// TIA Portal V20 export
DATA_BLOCK "CallEquipment_DB"   // DB76
{ DB_Accessible_From_OPC_UA := 'FALSE' }
// stored: AssignedProDiagFB Unit1.Em1.ProDiag, DBAccessibleFromOPCUA false, DBAccessibleFromWebserver false, InstanceOfName Unit1.Em1.CallEquipment, InstanceOfType FB, Namespace Unit1.Em1
"Unit1.Em1.CallEquipment"
   // VAR_INPUT
   //    ZoneOperationEnable { ExternalWritable := 'False'} : "LWONIK_typeSafetyZoneManualOperation";
   //    unitEnableControlInterfaces { ExternalWritable := 'False'} : "LAF_typeEnableControlInterfaces";
   //    commandExcute { ExternalWritable := 'False'} : Bool;
   // END_VAR
   // VAR_IN_OUT
   //    unitStatus : "LAF_typeUnitStatus";
   //    emFeedback : "LUC_typeEmFeedback";
   //    unitAlarmDB : "LAF_typeAlarms";
   // END_VAR
   // VAR
   //    instSequenceUnWinder { ExternalWritable := 'False'} : "Unit1.Em1.Sequence_1_UnWinder";
   //    instUnWinderInitializedJob1 { ExternalWritable := 'False'} : "LAF_SelectJob";
   //    instUnWinderRunJob2 { ExternalWritable := 'False'} : "LAF_SelectJob";
   //    instUnWinderStopJob3 { ExternalWritable := 'False'} : "LAF_SelectJob";
   //    instUnWinderRewindJob4 { ExternalWritable := 'False'} : "LAF_SelectJob";
   //    instCmUnWinderAxisB { ExternalWritable := 'False'} : "LBC_AxisControl_TecPlcCn";
   //    instCmAirShaftOnOff { ExternalWritable := 'False'} : "LBC_TwoWayActuatorCn";
   //    instcmExpelFwdBwd { ExternalWritable := 'False'} : "LBC_TwoWayActuatorCn";
   //    instCmTensionCheckSensor { ExternalWritable := 'False'} : "LBC_DigitalSignalCn";
   //    instCmRadiusMeasureAnalogInput { ExternalWritable := 'False'} : "LBC_AnalogInputCn";
   //    instCmEpc { ExternalWritable := 'False'} : "LER_EPC_CON600";
   //    instCmRadiusMeasure { ExternalWritable := 'False'} : "LER_RadiusMeasure";
   //    instUnWinderAxisControlInterlockSummary { ExternalWritable := 'False'} : "LER_AxisControl_InterlockSummary";
   //    instServoTorqueCal_DR2 { ExternalWritable := 'False'} : "LER_ServoTorqueCal";
   //    instLDrv701ControlUnWinderAxisB { ExternalWritable := 'False'} : "LDrvSafe_SinaTlg701Control";
   //    instLDrv701StatusUnWinderAxisB { ExternalWritable := 'False'} : "LDrvSafe_SinaTlg701Status";
   //    statUnitStatus { ExternalWritable := 'False'} : "LAF_typeUnitStatus";
   //    statAllBrakeTest { ExternalWritable := 'False'} : "LER_typeBrakeTestUnitCommands";
   //    instManageAlarms { ExternalWritable := 'False'} : "LAF_ManageAlarms";
   //    instEventsPFE { S7_SetPoint := 'True'} : "Unit1.Em1.EventsPFE";
   //    statEnableManualCmds { ExternalWritable := 'False'} : Bool;
   //    statRcEnableCmds { ExternalWritable := 'False'} : Bool;
   //    statPulse { ExternalWritable := 'False'} : Array[0..99] of Bool;
   //    statTonTimer { ExternalWritable := 'False'} : Array[0..99] of TON_TIME;
   //    statTofTimer { ExternalWritable := 'False'} : Array[0..99] of TOF_TIME;
   //    statRadius { ExternalWritable := 'False'} : LReal;
   //    statDiameter { ExternalWritable := 'False'} : LReal;
   //    citi_Ptrig : Array[0..20] of Bool;
   //    citiTon : Array[0..20] of TON_TIME;
   //    citi : Time;
   //    citiTest : Array[0..20] of Bool;
   //    SpeedLimitByRadius_Instance { S7_SetPoint := 'True'} : "Unit1.Em1.SpeedLimitByRadius";
   //    SpeedLimit { S7_SetPoint := 'True'} : LReal;
   //    SpeedRef : LReal;
   // END_VAR
BEGIN
END_DATA_BLOCK
